{attribute addProperty BoxType "CU1123-0010-0016"}
{attribute addProperty Id "A_0003_CU1124_0000_0016A_0003_CU1124_0000_0016_4FB9C66F992124"}
{attribute addProperty CRC "338944286"}
{attribute addProperty SizeInBites "992"}
{attribute addProperty SizeInBytes "124"}
TYPE A_0002_CU1123_0010_0016_1433E11E EXTENDS CU1123_179A0949 :
STRUCT
	{attribute addProperty Name "A_0003_CU1124_0000_0016"}
	A_0003_CU1124_0000_0016 : A_0003_CU1124_0000_0016_4FB9C66F;
END_STRUCT
END_TYPE

(* stored: Version 1.2.0.0, ProductVersion 3.1.4024.9
   DUT A_0002_CU1123_0010_0016_1433E11E: Id {49ba98e8-1cbd-4b3e-ba9e-1841d387c937} *)
